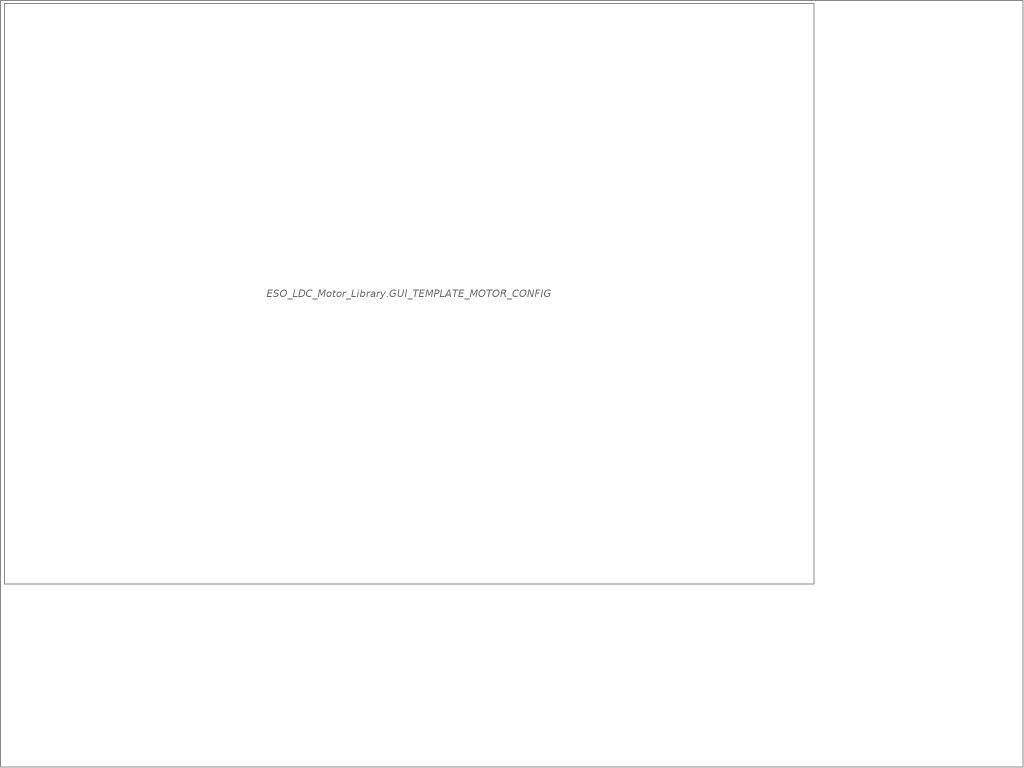
VISUALIZATION DL_Servo_1_Config  // 1024x768
    Frame (4,3 810x581)
        shows ESO_LDC_Motor_Library.GUI_TEMPLATE_MOTOR_CONFIG(m_Instance := MAIN.DL_Servo_1)
END_VISUALIZATION

(* stored: Version 1.1.0.1, ProductVersion 3.1.4024.12
   Visu DL_Servo_1_Config: Id {da63e479-ca1f-4a08-8165-b2e2c544b9d0} *)
